PROGRAM WebHmi
VAR
	watchDog1 : TON;
	watchDog2 : TON;
END_VAR

WatchDog();



hmi.Jog_Speed := Hmi_Web.Jog_Speed;

ACTION Clamp:

END_ACTION

ACTION WatchDog:
watchDog1(IN := NOT watchDog2.Q, PT:= T#500MS);
watchDog2(IN := watchDog1.Q, PT:= T#500MS);

Hmi_Web.Watchdog_Out := watchDog1.q;
END_ACTION

END_PROGRAM

(* stored: Version 1.1.0.1, ProductVersion 3.1.4026.13
   POU WebHmi: Id {7d27227b-25bd-493c-af6d-5b01257b715e}, SpecialFunc None
   Action Clamp: Id {6e3df157-7972-4f49-b719-7172aaa8a34f}
   Action WatchDog: Id {8d35982f-38a0-4f62-af87-136a45b979d4} *)
